// TIA Portal V20 export
DATA_BLOCK "EmData"   // DB40117
// stored: Access Published, MemoryReserve 100, Namespace Unit1
   VAR
      partData { S7_SetPoint := 'True'} : Array[0..14] of "LER_typePartData";
   END_VAR
BEGIN
   // partData[0] : jrOutPnPLeft
   // partData[1] : jrOutPnPRight
   // partData[2] : topTape
   // partData[3] : sideTape
   // partData[4] : transferPnPLeft
   // partData[5] : transferPnPRight
   // partData[6] : hotPressLeft
   // partData[7] : hotPressRight
   // partData[8] : hipotThickness
   // partData[9] : vision
   // partData[10] : laserMark
   // partData[11] : weightCheck
   // partData[12] : jrUnloadingPnP
   // partData[13] : StackNgBox
   // partData[14] : ConveryorA
END_DATA_BLOCK
